FUNCTION STATUS_TO_ESR : esr_data
VAR_INPUT
	status : BYTE;
	adress : STRING(10);
	DT_in : DT;
	TS : TIME;
END_VAR


(*
version 1.0	6 oct 2006
programmer 	hugo
tested by		tobias

status_to_esr creates esr data from a status byte.

*)

IF status < 100 THEN
	status_to_ESR.typ := 1;
ELSIF status < 200 THEN
	status_to_ESR.typ := 2;
ELSE
	status_to_ESR.typ := 3;
END_IF;
status_to_ESR.adress:= adress;
status_to_ESR.DS := DT_in;
status_to_ESR.TS := TS;
status_to_ESR.data[0] := status;

END_FUNCTION

(* stored: Version 1.1.0.1, ProductVersion 3.1.4022.7
   POU STATUS_TO_ESR: Id {c96338a4-c4c9-465e-90cf-053e5889aa84}, SpecialFunc None *)
